// TIA Portal V20 export
TYPE "LER_typeTrcvUDT"
// stored: Access Published
   STRUCT
      Input : Struct
         Enable : Bool;
         Cont : Bool;
         Len : UDInt;
         Adhoc : Bool;
      END_STRUCT;
      Output : Struct
         Done : Bool;
         Busy : Bool;
         Error : Bool;
         Status : Word;
         RcvLen : UDInt;
      END_STRUCT;
      InOut : Struct
         rfidData : Array[0..311] of Byte;
         ADDR : Bool;
         COM_RST : Bool;
      END_STRUCT;
   END_STRUCT;
END_TYPE
